{attribute 'qualified_only'}
VAR_GLOBAL CONSTANT
	MAX_NUMBER_OF_BUTTON_IN_MENU	: INT := 20;
	
END_VAR

(* stored: Version 1.1.0.1
   GVL GVL_HMIEConstans: Id {8f5771d4-0142-4111-9a81-ac5cf3458a4b} *)
